(* IEC 61131-3 sources: Lasal/CPU_5344_V01/Class/MPScontrolMessage, 1 file *)

(* ---- MPScontrolMessage.st ---- *)
(*!
<Class
	Name               = "MPScontrolMessage"
	Revision           = "0.0"
	RealtimeTask       = "false"
	CyclicTask         = "false"
	BackgroundTask     = "false"
	Sigmatek           = "false"
	OSInterface        = "false"
	HighPriority       = "false"
	Automatic          = "false"
	UpdateMode         = "Prescan"
	SharedCommandTable = "true"
	Objectsize         = "(420,360)">
	<Channels>
		<Server Name="ClassSvr" Visualized="false" Initialize="false" WriteProtected="true" Retentive="false"/>
		<Server Name="Data" Class="String" Visualized="true" Remotely="true" Initialize="true" WriteProtected="false" Retentive="false" Comment="use this channel to access the string functions"/>
		<Server Name="responseTag" Visualized="true" Initialize="false" WriteProtected="false" Retentive="false"/>
		<Server Name="show" Visualized="true" Initialize="false" WriteProtected="false" Retentive="false"/>
		<Server Name="typeTag" Visualized="true" Initialize="false" WriteProtected="false" Retentive="false"/>
		<Client Name="text" Required="true" Internal="true"/>
	</Channels>
	<Network Name="MPScontrolMessage">
		<!-- List of Components in this network -->
		<Components>
			<Object
				Name       = "text"
				Class      = "String"
				Position   = "(60,240)"
				Visualized = "true"
				Remotely   = "true">
				<Channels>
					<Server Name="Data"/>
					<Client Name="SingleRealloc" Value="1"/>
				</Channels>
			</Object>
		</Components>
		<Comments>
		</Comments>
		<!-- List of Connections in this network -->
		<Connections>
			<Connection Source="this.text" Destination="text.Data"/>
			<Connection Source="this.Data" Destination="text.Data" Vertices="(998,270),(826,330),"/>
		</Connections>
		<!-- Headerfiles -->
		<Options>
		</Options>
	</Network>
</Class>
*)
MPScontrolMessage : CLASS
  //Servers:
	ClassSvr 	: SvrChCmd_DINT;
	Data 	: SvrChCmd_UDINT;
	typeTag 	: SvrCh_DINT;
	responseTag 	: SvrCh_DINT;
	show 	: SvrCh_DINT;
  //Clients:
	text 	: CltChCmd_String;
  //Variables:
		tmpString 	: longText;
		isTheSame 	: DINT;
		len 	: UDINT;
  //Functions:

	FUNCTION GLOBAL showMessage
		VAR_INPUT
			string 	: longText;
			typeOffMessage 	: DINT;
		END_VAR;

	FUNCTION VIRTUAL GLOBAL Data::Read
		VAR_OUTPUT
			output (EAX) 	: UDINT;
		END_VAR;

	FUNCTION VIRTUAL GLOBAL Data::Write
		VAR_INPUT
			input (EAX) 	: UDINT;
		END_VAR
		VAR_OUTPUT
			result (EAX) 	: UDINT;
		END_VAR;

	FUNCTION VIRTUAL GLOBAL responseTag::Write
		VAR_INPUT
			input (EAX) 	: DINT;
		END_VAR
		VAR_OUTPUT
			result (EAX) 	: DINT;
		END_VAR;
  //Tables:
	FUNCTION @STD
		VAR_OUTPUT
			ret_code	: CONFSTATES;
		END_VAR;
	FUNCTION GLOBAL TAB @CT_;
END_CLASS;

#pragma using String

FUNCTION VIRTUAL GLOBAL MPScontrolMessage::Data::Read
	VAR_OUTPUT
		output (EAX) 	: UDINT;
	END_VAR

	Data := text.Data.Read();
	output := Data;

END_FUNCTION

FUNCTION VIRTUAL GLOBAL MPScontrolMessage::Data::Write
	VAR_INPUT
		input (EAX) 	: UDINT;
	END_VAR
	VAR_OUTPUT
		result (EAX) 	: UDINT;
	END_VAR

	Data := input;
	result := (text.Data.Write(Data))$UDINT;

END_FUNCTION

FUNCTION GLOBAL MPScontrolMessage::showMessage
	VAR_INPUT
		string 	: longText;
		typeOffMessage 	: DINT;
	END_VAR

  typeTag:= typeOffMessage; //can be 0 for ok message or 1 for yes/no

  responseTag:=0; //1 for yes, and -1 for no

  IF tmpString = string THEN
    isTheSame:= TRUE;
  ELSE
    isTheSame:= FALSE;
  END_IF;
  tmpString:= string;
  IF isTheSame THEN
    len:= _strlen(src:=#tmpString[0]);
    IF len <= 250 THEN
      tmpString[len]:= '.';
    END_IF;
  END_IF;
  show:= 1;
  text.WriteDataOff(udLen:=sizeof(longText), udOff:=0, pData:=#tmpString[0]);

END_FUNCTION

FUNCTION VIRTUAL GLOBAL MPScontrolMessage::responseTag::Write
	VAR_INPUT
		input (EAX) 	: DINT;
	END_VAR
	VAR_OUTPUT
		result (EAX) 	: DINT;
	END_VAR

	responseTag := input;
  show:= 0;
	result := responseTag;

END_FUNCTION
